TYPE ST_MemberAnounce :
STRUCT
	Laenge		:	WORD;
	receiver	:	WORD;
	Sender		:	WORD;
	Typ			:	WORD;
	Reserve		:	WORD;
	N_Laenge	:	WORD;
	Kommando	:	WORD;
END_STRUCT

END_TYPE

(* stored: Version 1.1.0.1, ProductVersion 3.1.4024.12
   DUT ST_MemberAnounce: Id {36ec1b87-9937-480d-8158-a78cf6705d38} *)
